PROGRAM PRG_VLS
VAR
    fbVLS_SLITS_TOP : FB_MotionStage;
    fbVLS_SLITS_BOTTOM : FB_MotionStage;
    fbVLS_SLITS_RIGHT : FB_MotionStage;
    fbVLS_SLITS_LEFT: FB_MotionStage;
    fbVLS_Mirror_P : FB_MotionStage;
    fbVLS_Grating_P : FB_MotionStage;
    fbVLS_CAM_P : FB_MotionStage;
    fbVLS_CAM_D : FB_MotionStage;

    bInit :BOOL:=TRUE;


    rGrating_Pitch :LREAL;
    rMirror_Pitch :LREAL;

END_VAR

IF ( bInit) THEN
    bInit := FALSE;
    //SLITS
    Main.M40.bHardwareEnable := TRUE;
    Main.M40.bPowerSelf :=TRUE;
    Main.M40.nBrakeMode := ENUM_StageBrakeMode.NO_BRAKE;
    Main.M40.nEnableMode := ENUM_StageEnableMode.DURING_MOTION;
    Main.M41.bHardwareEnable := TRUE;
    Main.M41.bPowerSelf :=TRUE;
    Main.M41.nBrakeMode := ENUM_StageBrakeMode.NO_BRAKE;
    Main.M41.nEnableMode := ENUM_StageEnableMode.DURING_MOTION;
    Main.M42.bHardwareEnable := TRUE;
    Main.M42.bPowerSelf :=TRUE;
    Main.M42.nBrakeMode := ENUM_StageBrakeMode.NO_BRAKE;
    Main.M42.nEnableMode := ENUM_StageEnableMode.DURING_MOTION;
    Main.M43.bHardwareEnable := TRUE;
    Main.M43.bPowerSelf :=TRUE;
    Main.M43.nBrakeMode := ENUM_StageBrakeMode.NO_BRAKE;
    Main.M43.nEnableMode := ENUM_StageEnableMode.DURING_MOTION;

    //Homing routine parameters
    Main.M40.fHomePosition:= 0;
    Main.M40.nHomingMode := ENUM_EpicsHomeCmd.LOW_LIMIT;
    Main.M41.fHomePosition:= 0;
    Main.M41.nHomingMode := ENUM_EpicsHomeCmd.LOW_LIMIT;
    Main.M42.fHomePosition:= 0;
    Main.M42.nHomingMode := ENUM_EpicsHomeCmd.LOW_LIMIT;
    Main.M43.fHomePosition:= 0;
    Main.M43.nHomingMode := ENUM_EpicsHomeCmd.LOW_LIMIT;

    //Focusing Mirror Pitch
    Main.M44.bHardwareEnable := TRUE;
    Main.M44.bPowerSelf :=TRUE;
    Main.M44.nBrakeMode := ENUM_StageBrakeMode.NO_BRAKE;
    Main.M44.nEnableMode := ENUM_StageEnableMode.DURING_MOTION;
    //Homing routine parameters
    Main.M44.fHomePosition:= -0.2288; // old homing position: -3.473;
    Main.M44.nHomingMode := ENUM_EpicsHomeCmd.LOW_LIMIT;

    //Grating Pitch
    Main.M45.bHardwareEnable := TRUE;
    Main.M45.bPowerSelf :=TRUE;
    Main.M45.nBrakeMode := ENUM_StageBrakeMode.NO_BRAKE;
    Main.M45.nEnableMode := ENUM_StageEnableMode.DURING_MOTION;
    //Homing routine parameters
    Main.M45.fHomePosition:= -1.74;
    Main.M45.nHomingMode := ENUM_EpicsHomeCmd.LOW_LIMIT;

    //Cam
    Main.M46.bHardwareEnable := TRUE;
    Main.M46.bPowerSelf :=TRUE;
    Main.M46.nBrakeMode := ENUM_StageBrakeMode.NO_BRAKE;
    Main.M46.nEnableMode := ENUM_StageEnableMode.DURING_MOTION;
    Main.M47.bHardwareEnable := TRUE;
    Main.M47.bPowerSelf :=TRUE;
    Main.M47.nBrakeMode := ENUM_StageBrakeMode.NO_BRAKE;
    Main.M47.nEnableMode := ENUM_StageEnableMode.DURING_MOTION;
    //Homing routine parameters
    Main.M46.fHomePosition:= 0.8923;
    Main.M46.nHomingMode := ENUM_EpicsHomeCmd.HIGH_LIMIT;//0 where it is horizontal
    Main.M47.fHomePosition:= -15.5;
    Main.M47.nHomingMode := ENUM_EpicsHomeCmd.LOW_LIMIT;
END_IF


//Calculate the mirror and grating pitch values
//OLD EQUATION:
//Mirror Pitch (x)  =   33.85 + 18.09x  - 0.2479x2
//rMirror_Pitch :=33.85 + (18.09*Main.M44.stAxisStatus.fActPosition(*mm*)  )- (0.2479 * EXPT(Main.M44.stAxisStatus.fActPosition,2));

//NEW EQUATION:
rMirror_Pitch :=27.667 + (18.1*Main.M44.stAxisStatus.fActPosition(*mm*)  )+ (-0.7569 * EXPT(Main.M44.stAxisStatus.fActPosition,2));

//Grating Pitch (x) =  22.56 - 16.25x + 0.334x2
rGrating_Pitch := 22.56 - (16.25*Main.M45.stAxisStatus.fActPosition(*mm*)  )+ (0.334 * EXPT(Main.M45.stAxisStatus.fActPosition,2));




fbVLS_SLITS_TOP(stMotionStage:=Main.M40);
fbVLS_SLITS_BOTTOM(stMotionStage:=Main.M41);
fbVLS_SLITS_RIGHT(stMotionStage:=Main.M42);
fbVLS_SLITS_LEFT(stMotionStage:=Main.M43);
fbVLS_Mirror_P(stMotionStage:=Main.M44);
fbVLS_Grating_P(stMotionStage:=Main.M45);
fbVLS_CAM_P(stMotionStage:=Main.M46);
fbVLS_CAM_D(stMotionStage:=Main.M47);

END_PROGRAM

(* stored: Version 1.1.0.1, ProductVersion 3.1.4022.18
   POU PRG_VLS: Id {89917009-bc34-43cd-b91a-9af045d34f25}, SpecialFunc None *)
